// Mitsubishi GX Works2 project: vision1007   PLC: Q02/Q02H

PROGRAM MAIN
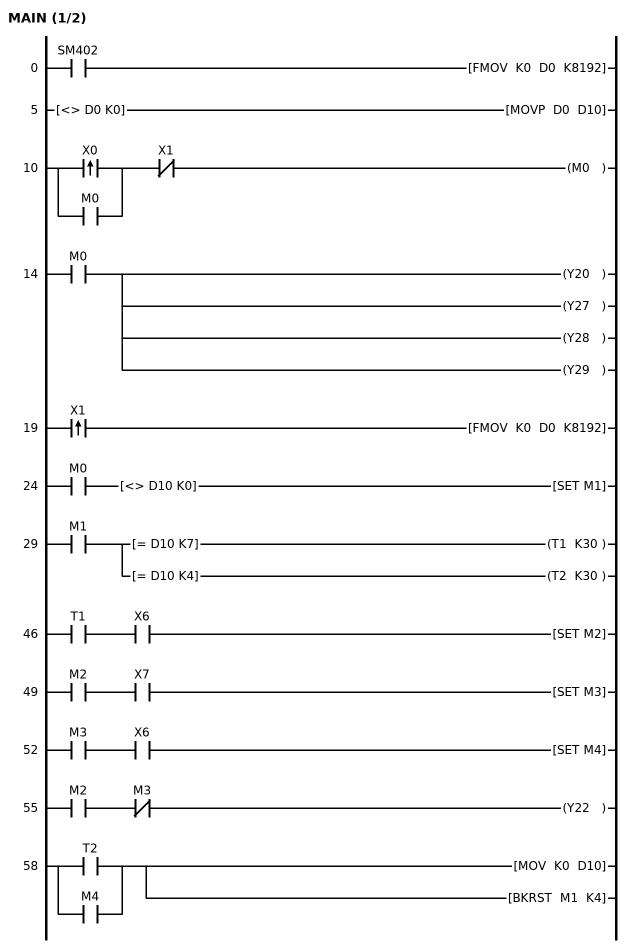
0     LD      SM402
      FMOV    K0 D0 K8192
5     LD<>    D0 K0
      MOVP    D0 D10
10    LDP     X0
      OR      M0
      ANI     X1
      OUT     M0
14    LD      M0
      OUT     Y20
      OUT     Y27
      OUT     Y28
      OUT     Y29
19    LDP     X1
      FMOV    K0 D0 K8192
24    LD      M0
      AND<>   D10 K0
      SET     M1
29    LD      M1
      MPS
      AND=    D10 K7
      OUT     T1 K30
      MPP
      AND=    D10 K4
      OUT     T2 K30
46    LD      T1
      AND     X6
      SET     M2
49    LD      M2
      AND     X7
      SET     M3
52    LD      M3
      AND     X6
      SET     M4
55    LD      M2
      ANI     M3
      OUT     Y22
58    LD      T2
      OR      M4
      MOV     K0 D10
      BKRST   M1 K4
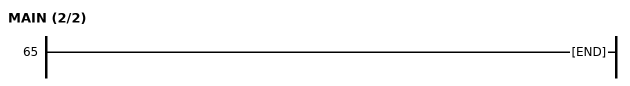
65    END
END_PROGRAM
